FUNCTION_BLOCK Gebhardt_Power
VAR_INPUT
	EN: BOOL;
	ModbusRTU: REFERENCE TO ModbusRTU;
	Address: BYTE := 101;
END_VAR
VAR_OUTPUT
	ENO: BOOL;
	Power: LREAL;
END_VAR
VAR
	ModbusWord_T_Power: ModbusReadWord;
END_VAR
VAR // added by the converter: edge detectors and wires of the graphical bodies
    _w1 : LREAL;
END_VAR

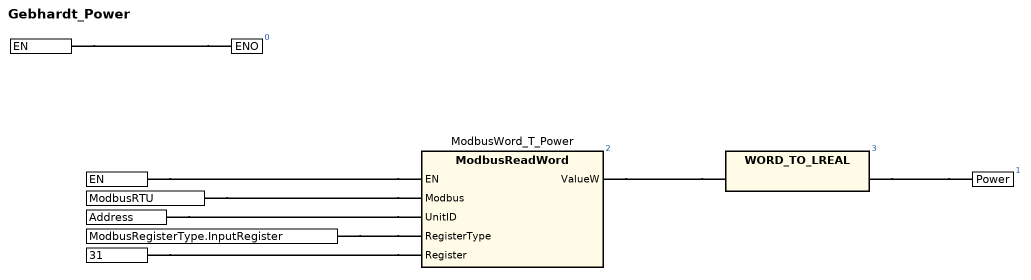
ENO := EN;
Power := _w1;
ModbusWord_T_Power(
    EN := EN,
    Modbus := ModbusRTU,
    UnitID := Address,
    RegisterType := ModbusRegisterType.InputRegister,
    Register := 31); // ModbusReadWord
_w1 := WORD_TO_LREAL(ModbusWord_T_Power.ValueW);

END_FUNCTION_BLOCK

(* stored: Version 1.1.0.1, ProductVersion 3.1.4024.6
   POU Gebhardt_Power: Id {9f827840-a2c2-4a9c-852c-4519fea070d1}, SpecialFunc None *)
